TYPE CoeSerialComSettings :
STRUCT
	IndexComPort1 : STRING;
	IndexComPort2 : STRING;
	EnableRtsCts : EnableRtsCts;
	EnableXonXoffTx : EnableXonXoffTx;
	EnableXonXoffRx : EnableXonXoffRx;
	BaudRate : BaudRate;
	DataFrame : DataFrame;
END_STRUCT
END_TYPE

(* stored: Version 1.1.0.1, ProductVersion 3.1.4024.3
   DUT CoeSerialComSettings: Id {b302206f-3262-4571-b2d7-71fdb0e488ed} *)
